// TIA Portal V19 export
FUNCTION "REGENRATION PROCESS" : Void   // FC14, LAD
{ S7_Optimized_Access := 'TRUE' }
// stored: SetENOAutomatically false
BEGIN

REGION Network 2: START PROCESS
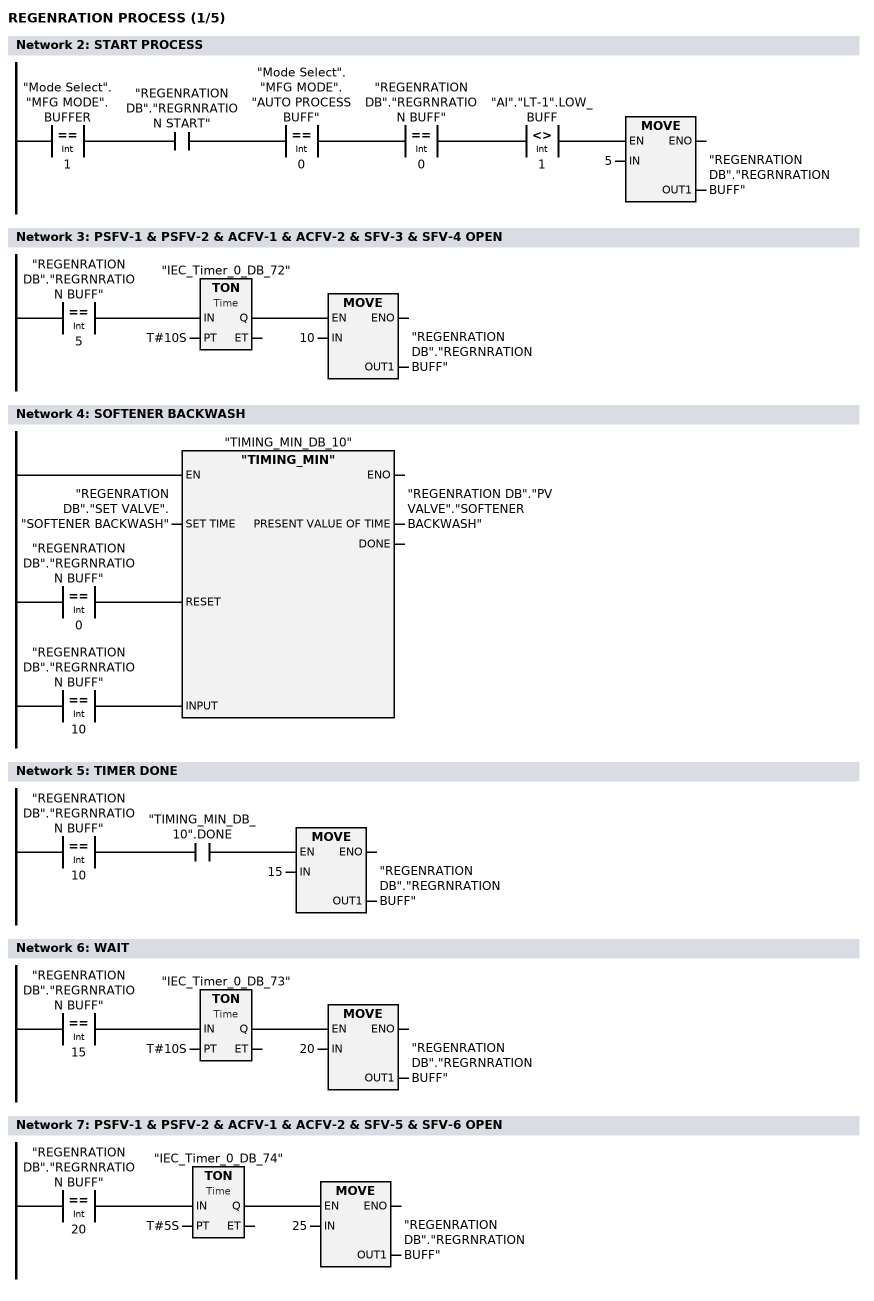
   RUNG wire#powerrail
      { S7_Templates := "SrcType := Int" } EQ_Contact(in1 := "Mode Select"."MFG MODE".BUFFER, in2 := 1)
      Contact( "REGENRATION DB"."REGRNRATION START" )
      { S7_Templates := "SrcType := Int" } EQ_Contact(in1 := "Mode Select"."MFG MODE"."AUTO PROCESS BUFF", in2 := 0)
      { S7_Templates := "SrcType := Int" } EQ_Contact(in1 := "REGENRATION DB"."REGRNRATION BUFF", in2 := 0)
      { S7_Templates := "SrcType := Int" } NE_Contact(in1 := "AI"."LT-1".LOW_BUFF, in2 := 1)
      Move(in := 5, out1 => "REGENRATION DB"."REGRNRATION BUFF")
   END_RUNG
   // the same network as SCL:
   IF ("Mode Select"."MFG MODE".BUFFER = 1) AND "REGENRATION DB"."REGRNRATION START" AND ("Mode Select"."MFG MODE"."AUTO PROCESS BUFF" = 0) AND ("REGENRATION DB"."REGRNRATION BUFF" = 0) AND ("AI"."LT-1".LOW_BUFF <> 1) THEN
       "REGENRATION DB"."REGRNRATION BUFF" := 5;
   END_IF;
END_REGION

REGION Network 3: PSFV-1 & PSFV-2 & ACFV-1 & ACFV-2 & SFV-3 & SFV-4 OPEN
   RUNG wire#powerrail
      { S7_Templates := "SrcType := Int" } EQ_Contact(in1 := "REGENRATION DB"."REGRNRATION BUFF", in2 := 5)
      { S7_Templates := "time_type := Time" } "IEC_Timer_0_DB_72".TON(pt := T#10S, et =>)
      Move(in := 10, out1 => "REGENRATION DB"."REGRNRATION BUFF")
   END_RUNG
   // the same network as SCL:
   "IEC_Timer_0_DB_72".TON(IN := "REGENRATION DB"."REGRNRATION BUFF" = 5, PT := T#10S);
   IF "IEC_Timer_0_DB_72".Q THEN "REGENRATION DB"."REGRNRATION BUFF" := 10; END_IF;
END_REGION

REGION Network 4: SOFTENER BACKWASH
   RUNG wire#powerrail
      "TIMING_MIN_DB_10"(RESET := wire#w1, INPUT := wire#w2, "SET TIME" := "REGENRATION DB"."SET VALVE"."SOFTENER BACKWASH", "PRESENT VALUE OF TIME" => "REGENRATION DB"."PV VALVE"."SOFTENER BACKWASH", DONE =>)
   END_RUNG
   RUNG wire#powerrail
      { S7_Templates := "SrcType := Int" } EQ_Contact(in1 := "REGENRATION DB"."REGRNRATION BUFF", in2 := 0)
   END_RUNG wire#w1
   RUNG wire#powerrail
      { S7_Templates := "SrcType := Int" } EQ_Contact(in1 := "REGENRATION DB"."REGRNRATION BUFF", in2 := 10)
   END_RUNG wire#w2
   // the same network as SCL:
   "TIMING_MIN_DB_10"("SET TIME" := "REGENRATION DB"."SET VALVE"."SOFTENER BACKWASH",   // "TIMING_MIN"
                      RESET := "REGENRATION DB"."REGRNRATION BUFF" = 0,
                      INPUT := "REGENRATION DB"."REGRNRATION BUFF" = 10,
                      "PRESENT VALUE OF TIME" => "REGENRATION DB"."PV VALVE"."SOFTENER BACKWASH");
END_REGION

REGION Network 5: TIMER DONE
   RUNG wire#powerrail
      { S7_Templates := "SrcType := Int" } EQ_Contact(in1 := "REGENRATION DB"."REGRNRATION BUFF", in2 := 10)
      Contact( "TIMING_MIN_DB_10".DONE )
      Move(in := 15, out1 => "REGENRATION DB"."REGRNRATION BUFF")
   END_RUNG
   // the same network as SCL:
   IF ("REGENRATION DB"."REGRNRATION BUFF" = 10) AND "TIMING_MIN_DB_10".DONE THEN
       "REGENRATION DB"."REGRNRATION BUFF" := 15;
   END_IF;
END_REGION

REGION Network 6: WAIT
   RUNG wire#powerrail
      { S7_Templates := "SrcType := Int" } EQ_Contact(in1 := "REGENRATION DB"."REGRNRATION BUFF", in2 := 15)
      { S7_Templates := "time_type := Time" } "IEC_Timer_0_DB_73".TON(pt := T#10S, et =>)
      Move(in := 20, out1 => "REGENRATION DB"."REGRNRATION BUFF")
   END_RUNG
   // the same network as SCL:
   "IEC_Timer_0_DB_73".TON(IN := "REGENRATION DB"."REGRNRATION BUFF" = 15, PT := T#10S);
   IF "IEC_Timer_0_DB_73".Q THEN "REGENRATION DB"."REGRNRATION BUFF" := 20; END_IF;
END_REGION

REGION Network 7: PSFV-1 & PSFV-2 & ACFV-1 & ACFV-2 & SFV-5 & SFV-6 OPEN
   RUNG wire#powerrail
      { S7_Templates := "SrcType := Int" } EQ_Contact(in1 := "REGENRATION DB"."REGRNRATION BUFF", in2 := 20)
      { S7_Templates := "time_type := Time" } "IEC_Timer_0_DB_74".TON(pt := T#5S, et =>)
      Move(in := 25, out1 => "REGENRATION DB"."REGRNRATION BUFF")
   END_RUNG
   // the same network as SCL:
   "IEC_Timer_0_DB_74".TON(IN := "REGENRATION DB"."REGRNRATION BUFF" = 20, PT := T#5S);
   IF "IEC_Timer_0_DB_74".Q THEN "REGENRATION DB"."REGRNRATION BUFF" := 25; END_IF;
END_REGION

REGION Network 8: SFV-3 & SFV-4 CLOSE
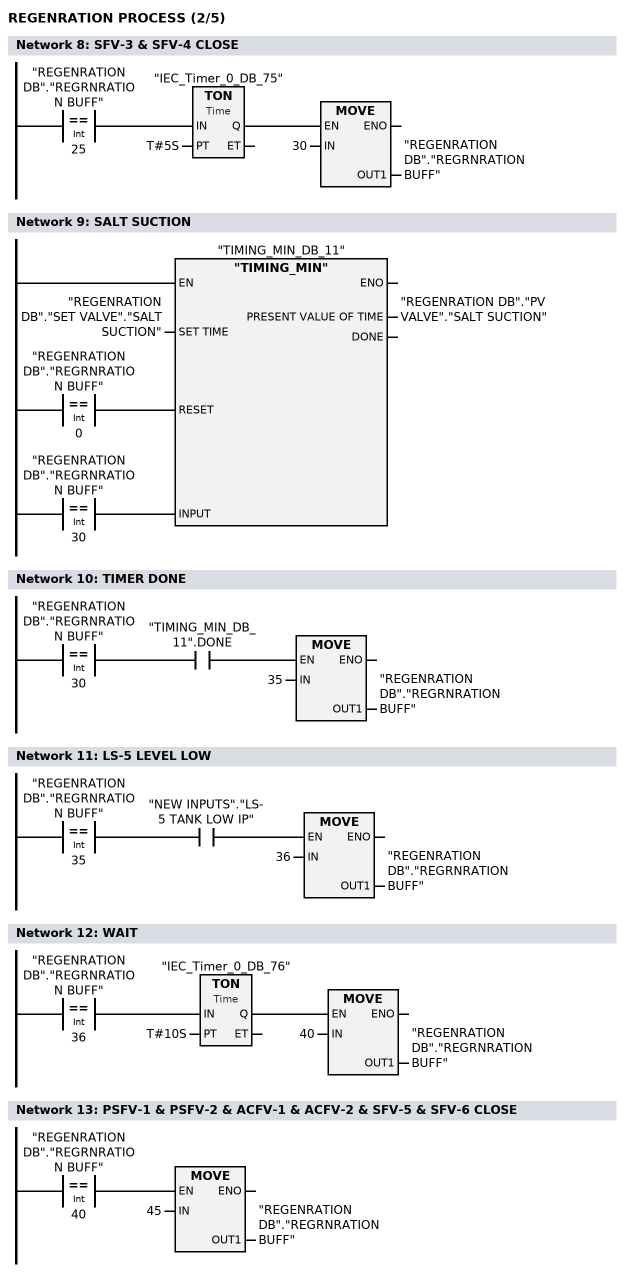
   RUNG wire#powerrail
      { S7_Templates := "SrcType := Int" } EQ_Contact(in1 := "REGENRATION DB"."REGRNRATION BUFF", in2 := 25)
      { S7_Templates := "time_type := Time" } "IEC_Timer_0_DB_75".TON(pt := T#5S, et =>)
      Move(in := 30, out1 => "REGENRATION DB"."REGRNRATION BUFF")
   END_RUNG
   // the same network as SCL:
   "IEC_Timer_0_DB_75".TON(IN := "REGENRATION DB"."REGRNRATION BUFF" = 25, PT := T#5S);
   IF "IEC_Timer_0_DB_75".Q THEN "REGENRATION DB"."REGRNRATION BUFF" := 30; END_IF;
END_REGION

REGION Network 9: SALT SUCTION
   RUNG wire#powerrail
      "TIMING_MIN_DB_11"(RESET := wire#w1, INPUT := wire#w2, "SET TIME" := "REGENRATION DB"."SET VALVE"."SALT SUCTION", "PRESENT VALUE OF TIME" => "REGENRATION DB"."PV VALVE"."SALT SUCTION", DONE =>)
   END_RUNG
   RUNG wire#powerrail
      { S7_Templates := "SrcType := Int" } EQ_Contact(in1 := "REGENRATION DB"."REGRNRATION BUFF", in2 := 0)
   END_RUNG wire#w1
   RUNG wire#powerrail
      { S7_Templates := "SrcType := Int" } EQ_Contact(in1 := "REGENRATION DB"."REGRNRATION BUFF", in2 := 30)
   END_RUNG wire#w2
   // the same network as SCL:
   "TIMING_MIN_DB_11"("SET TIME" := "REGENRATION DB"."SET VALVE"."SALT SUCTION",   // "TIMING_MIN"
                      RESET := "REGENRATION DB"."REGRNRATION BUFF" = 0,
                      INPUT := "REGENRATION DB"."REGRNRATION BUFF" = 30,
                      "PRESENT VALUE OF TIME" => "REGENRATION DB"."PV VALVE"."SALT SUCTION");
END_REGION

REGION Network 10: TIMER DONE
   RUNG wire#powerrail
      { S7_Templates := "SrcType := Int" } EQ_Contact(in1 := "REGENRATION DB"."REGRNRATION BUFF", in2 := 30)
      Contact( "TIMING_MIN_DB_11".DONE )
      Move(in := 35, out1 => "REGENRATION DB"."REGRNRATION BUFF")
   END_RUNG
   // the same network as SCL:
   IF ("REGENRATION DB"."REGRNRATION BUFF" = 30) AND "TIMING_MIN_DB_11".DONE THEN
       "REGENRATION DB"."REGRNRATION BUFF" := 35;
   END_IF;
END_REGION

REGION Network 11: LS-5 LEVEL LOW
   RUNG wire#powerrail
      { S7_Templates := "SrcType := Int" } EQ_Contact(in1 := "REGENRATION DB"."REGRNRATION BUFF", in2 := 35)
      Contact( "NEW INPUTS"."LS-5 TANK LOW IP" )
      Move(in := 36, out1 => "REGENRATION DB"."REGRNRATION BUFF")
   END_RUNG
   // the same network as SCL:
   IF ("REGENRATION DB"."REGRNRATION BUFF" = 35) AND "NEW INPUTS"."LS-5 TANK LOW IP" THEN
       "REGENRATION DB"."REGRNRATION BUFF" := 36;
   END_IF;
END_REGION

REGION Network 12: WAIT
   RUNG wire#powerrail
      { S7_Templates := "SrcType := Int" } EQ_Contact(in1 := "REGENRATION DB"."REGRNRATION BUFF", in2 := 36)
      { S7_Templates := "time_type := Time" } "IEC_Timer_0_DB_76".TON(pt := T#10S, et =>)
      Move(in := 40, out1 => "REGENRATION DB"."REGRNRATION BUFF")
   END_RUNG
   // the same network as SCL:
   "IEC_Timer_0_DB_76".TON(IN := "REGENRATION DB"."REGRNRATION BUFF" = 36, PT := T#10S);
   IF "IEC_Timer_0_DB_76".Q THEN "REGENRATION DB"."REGRNRATION BUFF" := 40; END_IF;
END_REGION

REGION Network 13: PSFV-1 & PSFV-2 & ACFV-1 & ACFV-2 & SFV-5 & SFV-6 CLOSE
   RUNG wire#powerrail
      { S7_Templates := "SrcType := Int" } EQ_Contact(in1 := "REGENRATION DB"."REGRNRATION BUFF", in2 := 40)
      Move(in := 45, out1 => "REGENRATION DB"."REGRNRATION BUFF")
   END_RUNG
   // the same network as SCL:
   IF "REGENRATION DB"."REGRNRATION BUFF" = 40 THEN "REGENRATION DB"."REGRNRATION BUFF" := 45; END_IF;
END_REGION

REGION Network 14: SALT HOLDING
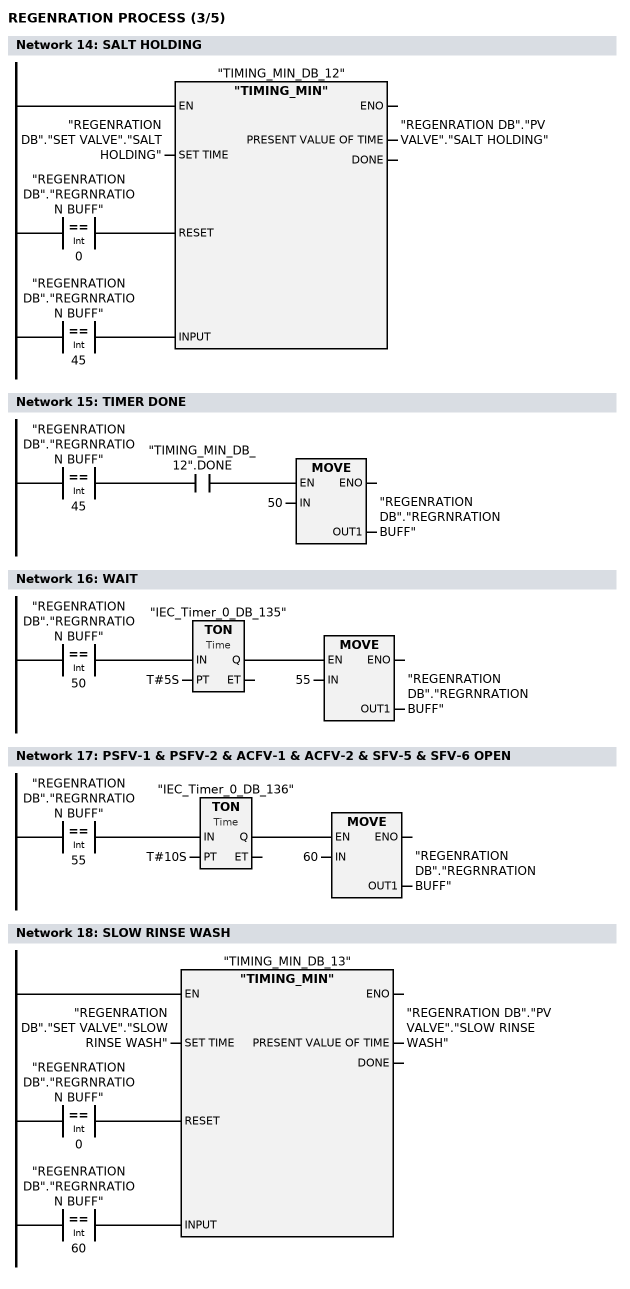
   RUNG wire#powerrail
      "TIMING_MIN_DB_12"(RESET := wire#w1, INPUT := wire#w2, "SET TIME" := "REGENRATION DB"."SET VALVE"."SALT HOLDING", "PRESENT VALUE OF TIME" => "REGENRATION DB"."PV VALVE"."SALT HOLDING", DONE =>)
   END_RUNG
   RUNG wire#powerrail
      { S7_Templates := "SrcType := Int" } EQ_Contact(in1 := "REGENRATION DB"."REGRNRATION BUFF", in2 := 0)
   END_RUNG wire#w1
   RUNG wire#powerrail
      { S7_Templates := "SrcType := Int" } EQ_Contact(in1 := "REGENRATION DB"."REGRNRATION BUFF", in2 := 45)
   END_RUNG wire#w2
   // the same network as SCL:
   "TIMING_MIN_DB_12"("SET TIME" := "REGENRATION DB"."SET VALVE"."SALT HOLDING",   // "TIMING_MIN"
                      RESET := "REGENRATION DB"."REGRNRATION BUFF" = 0,
                      INPUT := "REGENRATION DB"."REGRNRATION BUFF" = 45,
                      "PRESENT VALUE OF TIME" => "REGENRATION DB"."PV VALVE"."SALT HOLDING");
END_REGION

REGION Network 15: TIMER DONE
   RUNG wire#powerrail
      { S7_Templates := "SrcType := Int" } EQ_Contact(in1 := "REGENRATION DB"."REGRNRATION BUFF", in2 := 45)
      Contact( "TIMING_MIN_DB_12".DONE )
      Move(in := 50, out1 => "REGENRATION DB"."REGRNRATION BUFF")
   END_RUNG
   // the same network as SCL:
   IF ("REGENRATION DB"."REGRNRATION BUFF" = 45) AND "TIMING_MIN_DB_12".DONE THEN
       "REGENRATION DB"."REGRNRATION BUFF" := 50;
   END_IF;
END_REGION

REGION Network 16: WAIT
   RUNG wire#powerrail
      { S7_Templates := "SrcType := Int" } EQ_Contact(in1 := "REGENRATION DB"."REGRNRATION BUFF", in2 := 50)
      { S7_Templates := "time_type := Time" } "IEC_Timer_0_DB_135".TON(pt := T#5S, et =>)
      Move(in := 55, out1 => "REGENRATION DB"."REGRNRATION BUFF")
   END_RUNG
   // the same network as SCL:
   "IEC_Timer_0_DB_135".TON(IN := "REGENRATION DB"."REGRNRATION BUFF" = 50, PT := T#5S);
   IF "IEC_Timer_0_DB_135".Q THEN "REGENRATION DB"."REGRNRATION BUFF" := 55; END_IF;
END_REGION

REGION Network 17: PSFV-1 & PSFV-2 & ACFV-1 & ACFV-2 & SFV-5 & SFV-6 OPEN
   RUNG wire#powerrail
      { S7_Templates := "SrcType := Int" } EQ_Contact(in1 := "REGENRATION DB"."REGRNRATION BUFF", in2 := 55)
      { S7_Templates := "time_type := Time" } "IEC_Timer_0_DB_136".TON(pt := T#10S, et =>)
      Move(in := 60, out1 => "REGENRATION DB"."REGRNRATION BUFF")
   END_RUNG
   // the same network as SCL:
   "IEC_Timer_0_DB_136".TON(IN := "REGENRATION DB"."REGRNRATION BUFF" = 55, PT := T#10S);
   IF "IEC_Timer_0_DB_136".Q THEN "REGENRATION DB"."REGRNRATION BUFF" := 60; END_IF;
END_REGION

REGION Network 18: SLOW RINSE WASH
   RUNG wire#powerrail
      "TIMING_MIN_DB_13"(RESET := wire#w1, INPUT := wire#w2, "SET TIME" := "REGENRATION DB"."SET VALVE"."SLOW RINSE WASH", "PRESENT VALUE OF TIME" => "REGENRATION DB"."PV VALVE"."SLOW RINSE WASH", DONE =>)
   END_RUNG
   RUNG wire#powerrail
      { S7_Templates := "SrcType := Int" } EQ_Contact(in1 := "REGENRATION DB"."REGRNRATION BUFF", in2 := 0)
   END_RUNG wire#w1
   RUNG wire#powerrail
      { S7_Templates := "SrcType := Int" } EQ_Contact(in1 := "REGENRATION DB"."REGRNRATION BUFF", in2 := 60)
   END_RUNG wire#w2
   // the same network as SCL:
   "TIMING_MIN_DB_13"("SET TIME" := "REGENRATION DB"."SET VALVE"."SLOW RINSE WASH",   // "TIMING_MIN"
                      RESET := "REGENRATION DB"."REGRNRATION BUFF" = 0,
                      INPUT := "REGENRATION DB"."REGRNRATION BUFF" = 60,
                      "PRESENT VALUE OF TIME" => "REGENRATION DB"."PV VALVE"."SLOW RINSE WASH");
END_REGION

REGION Network 19: TIMER DONE
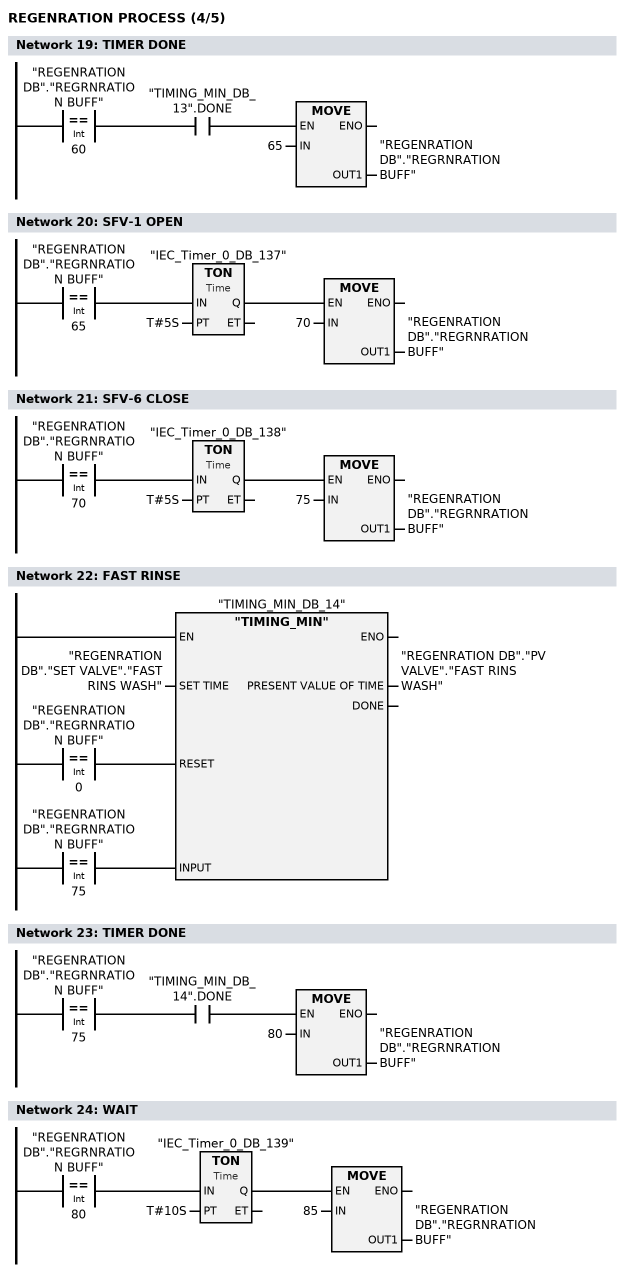
   RUNG wire#powerrail
      { S7_Templates := "SrcType := Int" } EQ_Contact(in1 := "REGENRATION DB"."REGRNRATION BUFF", in2 := 60)
      Contact( "TIMING_MIN_DB_13".DONE )
      Move(in := 65, out1 => "REGENRATION DB"."REGRNRATION BUFF")
   END_RUNG
   // the same network as SCL:
   IF ("REGENRATION DB"."REGRNRATION BUFF" = 60) AND "TIMING_MIN_DB_13".DONE THEN
       "REGENRATION DB"."REGRNRATION BUFF" := 65;
   END_IF;
END_REGION

REGION Network 20: SFV-1 OPEN
   RUNG wire#powerrail
      { S7_Templates := "SrcType := Int" } EQ_Contact(in1 := "REGENRATION DB"."REGRNRATION BUFF", in2 := 65)
      { S7_Templates := "time_type := Time" } "IEC_Timer_0_DB_137".TON(pt := T#5S, et =>)
      Move(in := 70, out1 => "REGENRATION DB"."REGRNRATION BUFF")
   END_RUNG
   // the same network as SCL:
   "IEC_Timer_0_DB_137".TON(IN := "REGENRATION DB"."REGRNRATION BUFF" = 65, PT := T#5S);
   IF "IEC_Timer_0_DB_137".Q THEN "REGENRATION DB"."REGRNRATION BUFF" := 70; END_IF;
END_REGION

REGION Network 21: SFV-6 CLOSE
   RUNG wire#powerrail
      { S7_Templates := "SrcType := Int" } EQ_Contact(in1 := "REGENRATION DB"."REGRNRATION BUFF", in2 := 70)
      { S7_Templates := "time_type := Time" } "IEC_Timer_0_DB_138".TON(pt := T#5S, et =>)
      Move(in := 75, out1 => "REGENRATION DB"."REGRNRATION BUFF")
   END_RUNG
   // the same network as SCL:
   "IEC_Timer_0_DB_138".TON(IN := "REGENRATION DB"."REGRNRATION BUFF" = 70, PT := T#5S);
   IF "IEC_Timer_0_DB_138".Q THEN "REGENRATION DB"."REGRNRATION BUFF" := 75; END_IF;
END_REGION

REGION Network 22: FAST RINSE
   RUNG wire#powerrail
      "TIMING_MIN_DB_14"(RESET := wire#w1, INPUT := wire#w2, "SET TIME" := "REGENRATION DB"."SET VALVE"."FAST RINS WASH", "PRESENT VALUE OF TIME" => "REGENRATION DB"."PV VALVE"."FAST RINS WASH", DONE =>)
   END_RUNG
   RUNG wire#powerrail
      { S7_Templates := "SrcType := Int" } EQ_Contact(in1 := "REGENRATION DB"."REGRNRATION BUFF", in2 := 0)
   END_RUNG wire#w1
   RUNG wire#powerrail
      { S7_Templates := "SrcType := Int" } EQ_Contact(in1 := "REGENRATION DB"."REGRNRATION BUFF", in2 := 75)
   END_RUNG wire#w2
   // the same network as SCL:
   "TIMING_MIN_DB_14"("SET TIME" := "REGENRATION DB"."SET VALVE"."FAST RINS WASH",   // "TIMING_MIN"
                      RESET := "REGENRATION DB"."REGRNRATION BUFF" = 0,
                      INPUT := "REGENRATION DB"."REGRNRATION BUFF" = 75,
                      "PRESENT VALUE OF TIME" => "REGENRATION DB"."PV VALVE"."FAST RINS WASH");
END_REGION

REGION Network 23: TIMER DONE
   RUNG wire#powerrail
      { S7_Templates := "SrcType := Int" } EQ_Contact(in1 := "REGENRATION DB"."REGRNRATION BUFF", in2 := 75)
      Contact( "TIMING_MIN_DB_14".DONE )
      Move(in := 80, out1 => "REGENRATION DB"."REGRNRATION BUFF")
   END_RUNG
   // the same network as SCL:
   IF ("REGENRATION DB"."REGRNRATION BUFF" = 75) AND "TIMING_MIN_DB_14".DONE THEN
       "REGENRATION DB"."REGRNRATION BUFF" := 80;
   END_IF;
END_REGION

REGION Network 24: WAIT
   RUNG wire#powerrail
      { S7_Templates := "SrcType := Int" } EQ_Contact(in1 := "REGENRATION DB"."REGRNRATION BUFF", in2 := 80)
      { S7_Templates := "time_type := Time" } "IEC_Timer_0_DB_139".TON(pt := T#10S, et =>)
      Move(in := 85, out1 => "REGENRATION DB"."REGRNRATION BUFF")
   END_RUNG
   // the same network as SCL:
   "IEC_Timer_0_DB_139".TON(IN := "REGENRATION DB"."REGRNRATION BUFF" = 80, PT := T#10S);
   IF "IEC_Timer_0_DB_139".Q THEN "REGENRATION DB"."REGRNRATION BUFF" := 85; END_IF;
END_REGION

REGION Network 25: PSFV-1 & PSFV-2 & ACFV-1 & ACFV-2 & SFV-5 & SFV-1 CLOSE
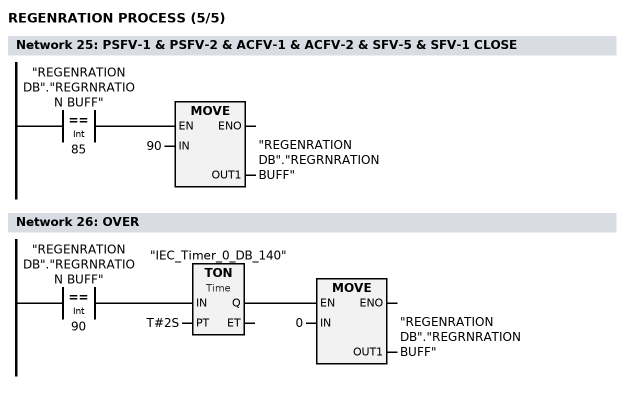
   RUNG wire#powerrail
      { S7_Templates := "SrcType := Int" } EQ_Contact(in1 := "REGENRATION DB"."REGRNRATION BUFF", in2 := 85)
      Move(in := 90, out1 => "REGENRATION DB"."REGRNRATION BUFF")
   END_RUNG
   // the same network as SCL:
   IF "REGENRATION DB"."REGRNRATION BUFF" = 85 THEN "REGENRATION DB"."REGRNRATION BUFF" := 90; END_IF;
END_REGION

REGION Network 26: OVER
   RUNG wire#powerrail
      { S7_Templates := "SrcType := Int" } EQ_Contact(in1 := "REGENRATION DB"."REGRNRATION BUFF", in2 := 90)
      { S7_Templates := "time_type := Time" } "IEC_Timer_0_DB_140".TON(pt := T#2S, et =>)
      Move(in := 0, out1 => "REGENRATION DB"."REGRNRATION BUFF")
   END_RUNG
   // the same network as SCL:
   "IEC_Timer_0_DB_140".TON(IN := "REGENRATION DB"."REGRNRATION BUFF" = 90, PT := T#2S);
   IF "IEC_Timer_0_DB_140".Q THEN "REGENRATION DB"."REGRNRATION BUFF" := 0; END_IF;
END_REGION
END_FUNCTION
